// TIA Portal V17 export
// export: Created 2026-01-01T00:00:00, ExportSetting WithDefaults, DisplayName synthetic-fixture, DisplayVersion machine-intelligence-v1.0.0
FUNCTION_BLOCK "FB_ConveyorCtrl"   // FB, SCL
BEGIN

NETWORK
TITLE = 
RunCmd := Start AND NOT Stop AND AutoMode AND Ready AND NOT Jam;

NETWORK
TITLE = 
FaultLamp := Jam OR NOT ProtectFb;
END_FUNCTION_BLOCK
